FUNCTION_BLOCK FB_Ethercat EXTENDS FB_Component
VAR_INPUT
    NetId 			AT %I*:		T_AmsNetIdArr;
	Slaves			AT %I*: 	UINT;
END_VAR
VAR_OUTPUT
END_VAR
VAR
	fbGetMasterState: 			FB_EcGetMasterDevState;
	fbMasterFrameStatistic:		FB_EcMasterFrameStatistic;
	fbGetSlaveStates:			FB_EcGetAllSlaveStates;
	pSlaveState:				POINTER TO Tc2_EtherCAT.ST_EcSlaveState;
END_VAR

METHOD PUBLIC M_Call
VAR_INPUT
END_VAR
SUPER^.M_Call();

fbGetMasterState(sNetId:= F_CreateAmsNetId(NetId));

fbMasterFrameStatistic(sNetId:= F_CreateAmsNetId(NetId));


IF pSlaveState = 0 THEN
		pSlaveState:= __NEW(BYTE, (SIZEOF(Tc2_EtherCAT.ST_EcSlaveState) * Slaves));
END_IF

fbGetSlaveStates(	sNetId:= F_CreateAmsNetId(NetId), 
					pStateBuf:= pSlaveState, 
					cbBufLen:= Slaves * SIZEOF(Tc2_EtherCAT.ST_EcSlaveState));
END_METHOD

END_FUNCTION_BLOCK

(* stored: Version 1.1.0.1, ProductVersion 3.1.4024.12
   POU FB_Ethercat: Id {26632774-44df-0f9a-1531-badc4b6ed605}, SpecialFunc None
   Method M_Call: Id {5844d1aa-3ea0-0990-1f38-2a22743f5d8b} *)
